(* Logix 5000 project; controller DUNEW2PLC1 vendor 1 type 14 code 221 rev 33.11; software revision 33.00; part 2 of 4 *)
(* tags used below, declared in another part *)
   LatchingTimeoutCounter : COUNTER;   // When you enter state 6 or 7, start counting seconds
   TimeoutTimer1 : TIMER;
   TimeoutTimer2 : TIMER;
   accel_xy : REAL;   // Tangential acceleration of the winding head in xy-plane
   ACTUATOR_POS : DINT;
   ALL_EOT_GOOD : BOOL;
   APA_IS_VERTICAL : BOOL;
   blink_off : TIMER;
   blink_on : TIMER;
   check_tension_stable : BOOL;   // Check if the tension is stable at the setpoint before moving the winding head
   ERROR_CODE : DINT;
   FRAME_LOC_FT_BTM : BOOL;
   FRAME_LOC_FT_MID : BOOL;
   FRAME_LOC_FT_TOP : BOOL;
   FRAME_LOC_HD_BTM : BOOL;
   FRAME_LOC_HD_MID : BOOL;
   FRAME_LOC_HD_TOP : BOOL;
   gamma : REAL;
   HEAD_POS : DINT;
   INIT_DONE : BOOL;
   J : REAL;
   MACHINE_SW_STAT : BOOL[32];
   MAS : BOOL;   // Motion Axis Stop
   MASTER_Z_GO : BOOL;
   MAX_TOLERABLE_Z : REAL;
   MCCD_X_Y_Axis1 : MOTION_INSTRUCTION;
   MINUS_X_EOT : BOOL;
   MINUS_Y_EOT : BOOL;
   MOVE_TYPE : INT;   // 0 = No Move 1 = XY JOG 2 = XY Plane Move 3 = Z JOG 4 = Z Axis Move 5 = Toggle Latch Actuator 6 = Home the Latch Actuator
   NEXTSTATE : DINT;
   PLUS_X_EOT : BOOL;
   PLUS_Y_EOT : BOOL;
   ResetPB : BOOL;
   Safety_Tripped_S : BOOL;
   speed_regulator_switch : BOOL;   // This is our "enable safe speed" switch, repurposed to switch the speed regulator
   STATE : DINT;   // CURRENT State Machine State
   T01 : TIMER;
   tension : ALIAS FOR Local:4:I.Ch01.Data;   // wire tension (N)
   TENSION_CONTROL_OK : BOOL;
   TENSION_ON_SWITCH : BOOL;
   tension_stable_timer : TIMER;
   v_0 : REAL;
   v_xy : REAL;   // velocity of winding head in xy plane
   v_xyz : REAL;   // Velocity of winding head in xyz space
   wire_break_proxy : BOOL;
   wire_break_tension : REAL;
   X_axis : AXIS_CIP_DRIVE;
   X_PARKED : BOOL;
   X_POSITION : ALIAS FOR POSITION[0,0];
   X_XFER_OK : BOOL;   // If at the head, check head support arms. Same for foot
   X_Y : COORDINATE_SYSTEM;
   XY_ACCELERATION : REAL;   // Maximum positive acceleration for position move.
   XY_DECELERATION : REAL;   // Maximum negative acceleration for position move.
   XY_SPEED : REAL;   // Maximum velocity for position move.
   XY_SPEED_REQ : REAL;   // XY Requested speed copy of XY_Speed to be used for MCLM and MCCD in MoveXY
   Y_axis : AXIS_CIP_DRIVE;
   Y_MOUNT_XFER_OK : BOOL;
   Y_POSITION : ALIAS FOR POSITION[0,1];
   Y_XFER_OK : BOOL;
   Y_Xfer_Window_Btm : BOOL;
   Y_Xfer_Window_Mid : BOOL;
   Y_Xfer_Window_Top : BOOL;
   Z_axis : AXIS_CIP_DRIVE;
   Z_EOT : BOOL;
   Z_EXTENDED : BOOL;
   Z_FIXED_LATCHED : BOOL;
   Z_FIXED_PRESENT : BOOL;
   Z_RETRACTED : BOOL;
   Z_STAGE_LATCHED : BOOL;
   Z_STAGE_PRESENT : BOOL;   // Winding head is on the Z-arm
(* Latch_UnLatch_State_6_7_8, continued *)

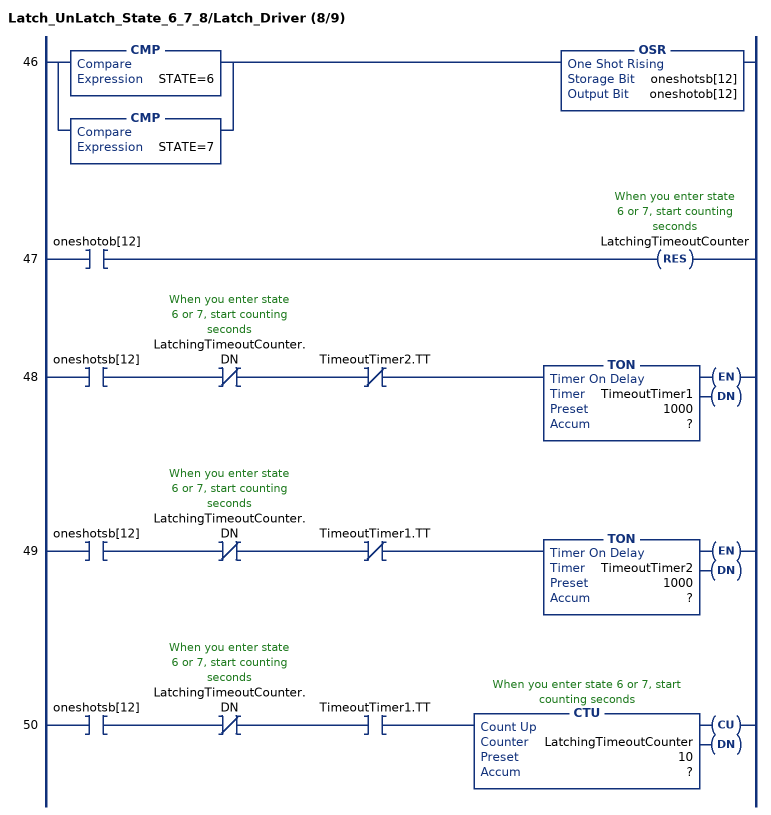
   [picture p24: Latch_UnLatch_State_6_7_8/Latch_Driver rungs 46-50]
   46: [CMP(STATE=6) ,CMP(STATE=7) ]OSR(oneshotsb[12],oneshotob[12]);
   47: XIC(oneshotob[12])RES(LatchingTimeoutCounter);
   48: XIC(oneshotsb[12])XIO(LatchingTimeoutCounter.DN)XIO(TimeoutTimer2.TT)TON(TimeoutTimer1,?,?);
   49: XIC(oneshotsb[12])XIO(LatchingTimeoutCounter.DN)XIO(TimeoutTimer1.TT)TON(TimeoutTimer2,?,?);
   50: XIC(oneshotsb[12])XIO(LatchingTimeoutCounter.DN)XIC(TimeoutTimer1.TT)CTU(LatchingTimeoutCounter,?,?);
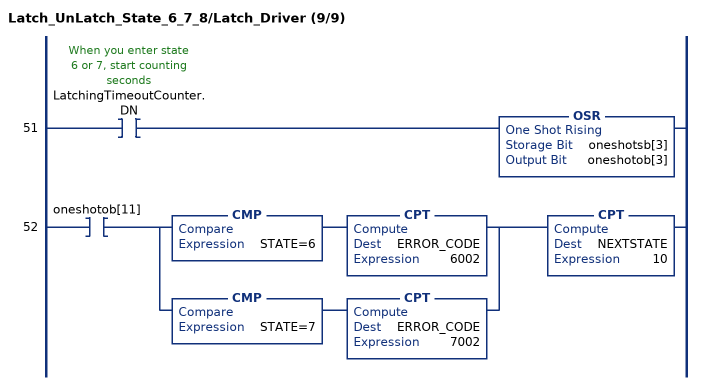
   51: XIC(LatchingTimeoutCounter.DN)OSR(oneshotsb[3],oneshotob[3]);
   52: XIC(oneshotob[11])[CMP(STATE=6) CPT(ERROR_CODE,6002) ,CMP(STATE=7) CPT(ERROR_CODE,7002) ]CPT(NEXTSTATE,10);
END_ROUTINE
END_PROGRAM

PROGRAM MainProgram   (* main routine MainRoutine *)
VAR
   Z_RETRACTED_1A : BOOL := 1; {access Read Only}
   Z_RETRACTED_1B : BOOL := 1; {access Read Only}
   Z_RETRACTED_2A : BOOL := 1; {access Read Only}
   Z_RETRACTED_2B : BOOL := 1; {access Read Only}
END_VAR

ROUTINE MainRoutine   (* ladder *)
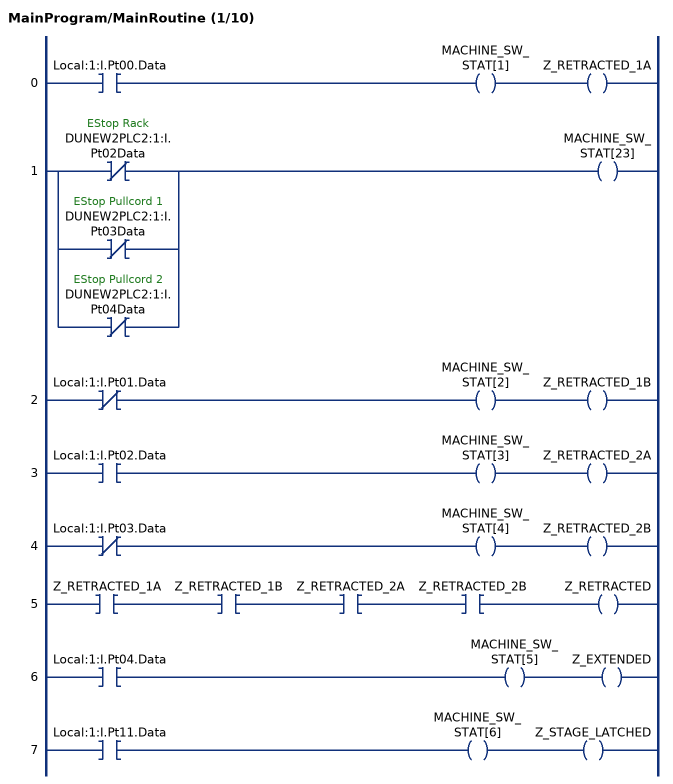
   0: XIC(Local:1:I.Pt00.Data)OTE(MACHINE_SW_STAT[1])OTE(Z_RETRACTED_1A);
   1: [XIO(DUNEW2PLC2:1:I.Pt02Data) ,[XIO(DUNEW2PLC2:1:I.Pt03Data) ,XIO(DUNEW2PLC2:1:I.Pt04Data) ] ]OTE(MACHINE_SW_STAT[23]);
   2: XIO(Local:1:I.Pt01.Data)OTE(MACHINE_SW_STAT[2])OTE(Z_RETRACTED_1B);
   3: XIC(Local:1:I.Pt02.Data)OTE(MACHINE_SW_STAT[3])OTE(Z_RETRACTED_2A);
   4: XIO(Local:1:I.Pt03.Data)OTE(MACHINE_SW_STAT[4])OTE(Z_RETRACTED_2B);
   5: XIC(Z_RETRACTED_1A)XIC(Z_RETRACTED_1B)XIC(Z_RETRACTED_2A)XIC(Z_RETRACTED_2B)OTE(Z_RETRACTED);
   6: XIC(Local:1:I.Pt04.Data)OTE(MACHINE_SW_STAT[5])OTE(Z_EXTENDED);
   7: XIC(Local:1:I.Pt11.Data)OTE(MACHINE_SW_STAT[6])OTE(Z_STAGE_LATCHED);
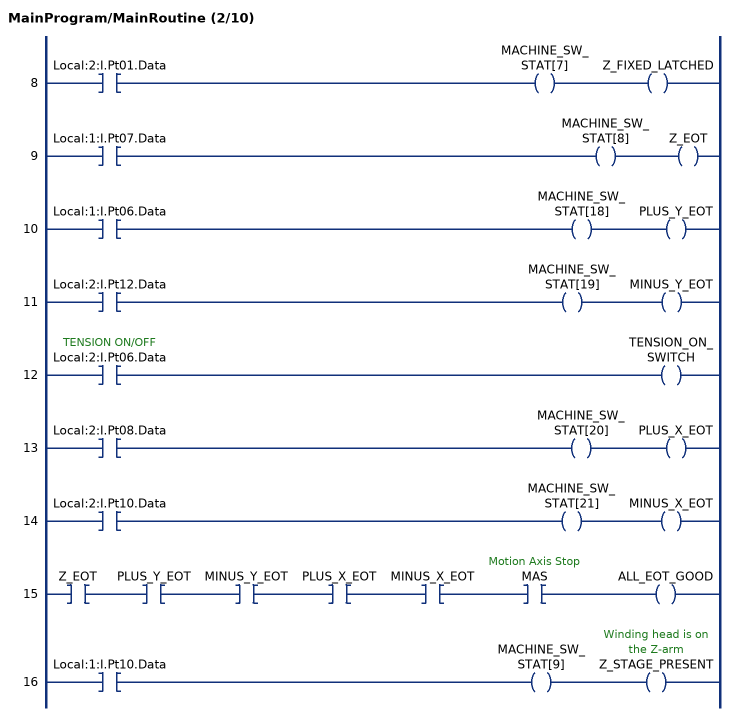
   8: XIC(Local:2:I.Pt01.Data)OTE(MACHINE_SW_STAT[7])OTE(Z_FIXED_LATCHED);
   9: XIC(Local:1:I.Pt07.Data)OTE(MACHINE_SW_STAT[8])OTE(Z_EOT);
   10: XIC(Local:1:I.Pt06.Data)OTE(MACHINE_SW_STAT[18])OTE(PLUS_Y_EOT);
   11: XIC(Local:2:I.Pt12.Data)OTE(MACHINE_SW_STAT[19])OTE(MINUS_Y_EOT);
   12: XIC(Local:2:I.Pt06.Data)OTE(TENSION_ON_SWITCH);
   13: XIC(Local:2:I.Pt08.Data)OTE(MACHINE_SW_STAT[20])OTE(PLUS_X_EOT);
   14: XIC(Local:2:I.Pt10.Data)OTE(MACHINE_SW_STAT[21])OTE(MINUS_X_EOT);
   15: XIC(Z_EOT)XIC(PLUS_Y_EOT)XIC(MINUS_Y_EOT)XIC(PLUS_X_EOT)XIC(MINUS_X_EOT)XIC(MAS)OTE(ALL_EOT_GOOD);
   16: XIC(Local:1:I.Pt10.Data)OTE(MACHINE_SW_STAT[9])OTE(Z_STAGE_PRESENT);
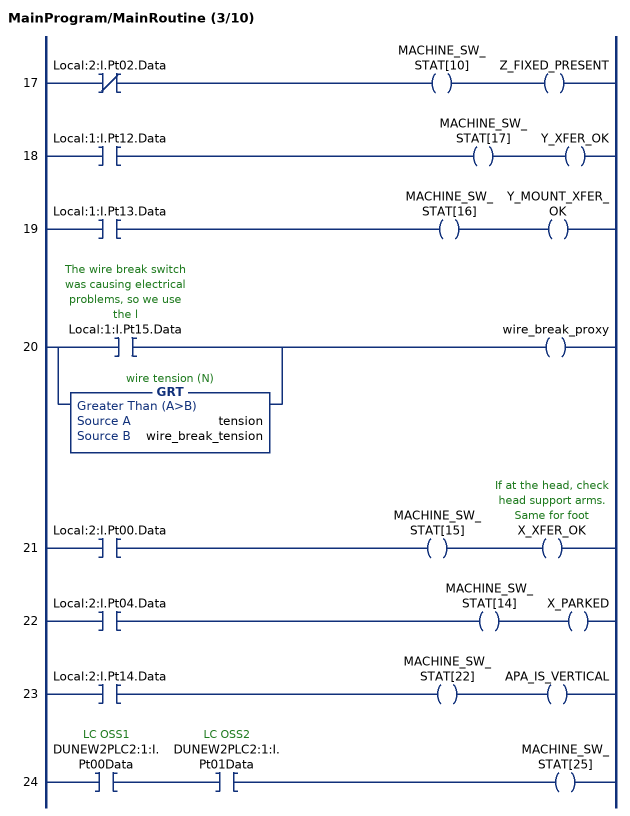
   17: XIO(Local:2:I.Pt02.Data)OTE(MACHINE_SW_STAT[10])OTE(Z_FIXED_PRESENT);
   18: XIC(Local:1:I.Pt12.Data)OTE(MACHINE_SW_STAT[17])OTE(Y_XFER_OK);
   19: XIC(Local:1:I.Pt13.Data)OTE(MACHINE_SW_STAT[16])OTE(Y_MOUNT_XFER_OK);
   20: [XIC(Local:1:I.Pt15.Data) ,GRT(tension,wire_break_tension) ]OTE(wire_break_proxy);
   21: XIC(Local:2:I.Pt00.Data)OTE(MACHINE_SW_STAT[15])OTE(X_XFER_OK);
   22: XIC(Local:2:I.Pt04.Data)OTE(MACHINE_SW_STAT[14])OTE(X_PARKED);
   23: XIC(Local:2:I.Pt14.Data)OTE(MACHINE_SW_STAT[22])OTE(APA_IS_VERTICAL);
   24: XIC(DUNEW2PLC2:1:I.Pt00Data)XIC(DUNEW2PLC2:1:I.Pt01Data)OTE(MACHINE_SW_STAT[25]);
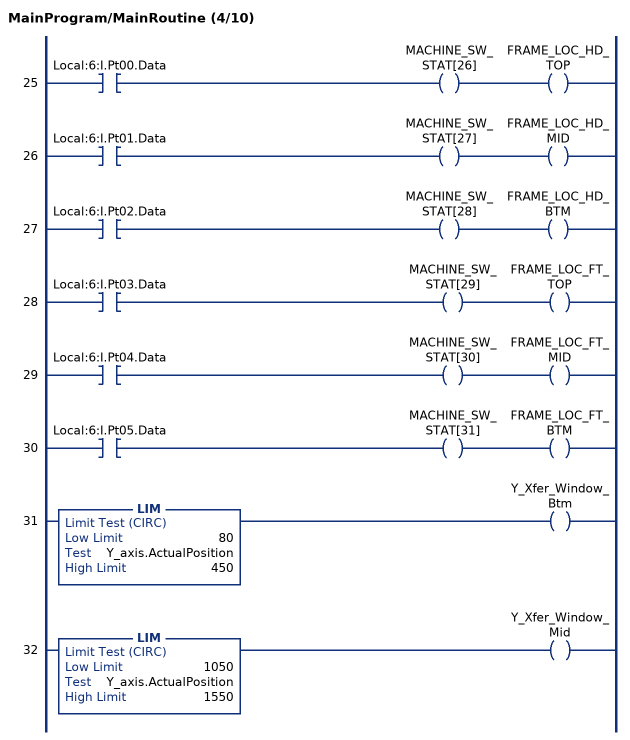
   25: XIC(Local:6:I.Pt00.Data)OTE(MACHINE_SW_STAT[26])OTE(FRAME_LOC_HD_TOP);
   26: XIC(Local:6:I.Pt01.Data)OTE(MACHINE_SW_STAT[27])OTE(FRAME_LOC_HD_MID);
   27: XIC(Local:6:I.Pt02.Data)OTE(MACHINE_SW_STAT[28])OTE(FRAME_LOC_HD_BTM);
   28: XIC(Local:6:I.Pt03.Data)OTE(MACHINE_SW_STAT[29])OTE(FRAME_LOC_FT_TOP);
   29: XIC(Local:6:I.Pt04.Data)OTE(MACHINE_SW_STAT[30])OTE(FRAME_LOC_FT_MID);
   30: XIC(Local:6:I.Pt05.Data)OTE(MACHINE_SW_STAT[31])OTE(FRAME_LOC_FT_BTM);
   31: LIM(80,Y_axis.ActualPosition,450)OTE(Y_Xfer_Window_Btm);
   32: LIM(1050,Y_axis.ActualPosition,1550)OTE(Y_Xfer_Window_Mid);
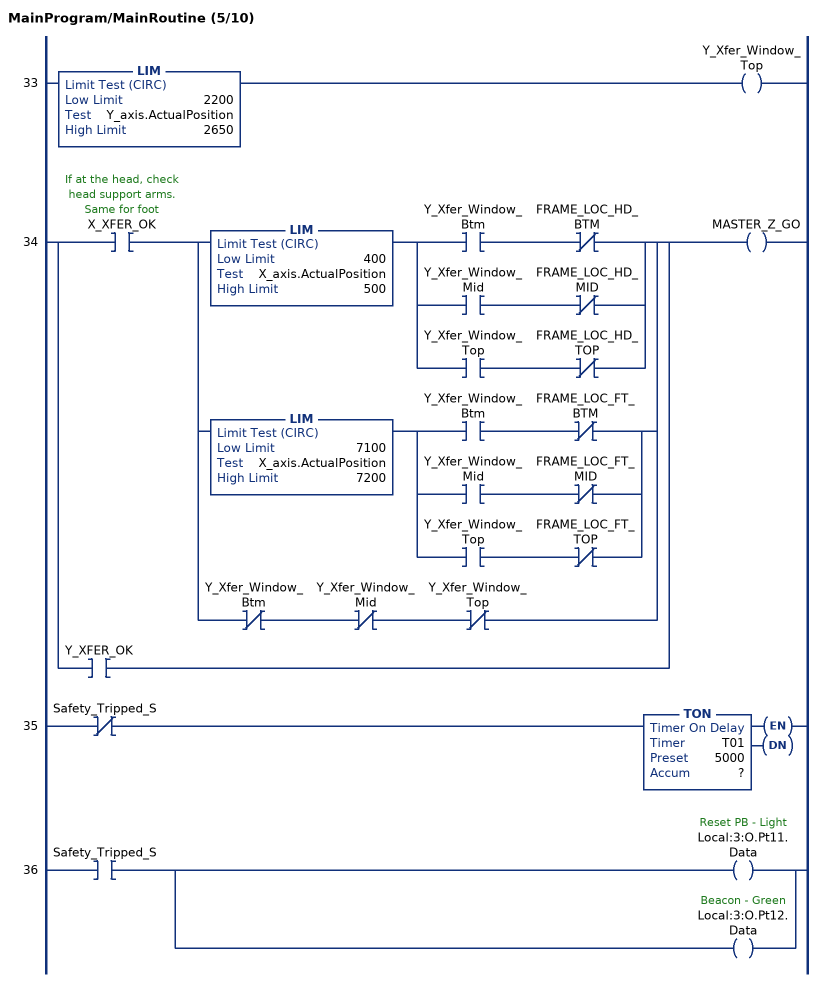
   33: LIM(2200,Y_axis.ActualPosition,2650)OTE(Y_Xfer_Window_Top);
   34: [XIC(X_XFER_OK) [LIM(400,X_axis.ActualPosition,500) [XIC(Y_Xfer_Window_Btm) XIO(FRAME_LOC_HD_BTM) ,XIC(Y_Xfer_Window_Mid) XIO(FRAME_LOC_HD_MID) ,XIC(Y_Xfer_Window_Top) XIO(FRAME_LOC_HD_TOP) ] ,LIM(7100,X_axis.ActualPosition,7200) [XIC(Y_Xfer_Window_Btm) XIO(FRAME_LOC_FT_BTM) ,XIC(Y_Xfer_Window_Mid) XIO(FRAME_LOC_FT_MID) ,XIC(Y_Xfer_Window_Top) XIO(FRAME_LOC_FT_TOP) ] ,XIO(Y_Xfer_Window_Btm) XIO(Y_Xfer_Window_Mid) XIO(Y_Xfer_Window_Top) ] ,XIC(Y_XFER_OK) ]OTE(MASTER_Z_GO);
   35: XIO(Safety_Tripped_S)TON(T01,?,?);
   36: XIC(Safety_Tripped_S)[OTE(Local:3:O.Pt11.Data) ,OTE(Local:3:O.Pt12.Data) ];
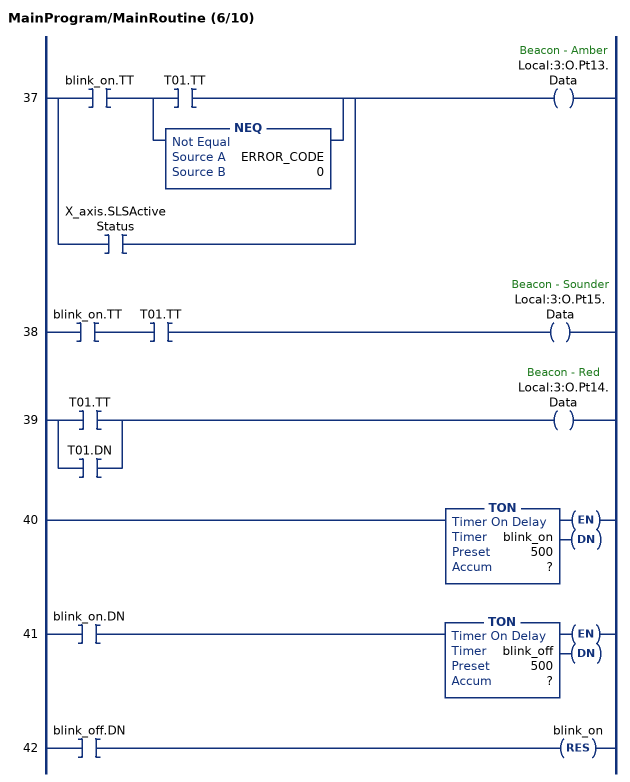
   37: [XIC(blink_on.TT) [XIC(T01.TT) ,NEQ(ERROR_CODE,0) ] ,XIC(X_axis.SLSActiveStatus) ]OTE(Local:3:O.Pt13.Data);
   38: XIC(blink_on.TT)XIC(T01.TT)OTE(Local:3:O.Pt15.Data);
   39: [XIC(T01.TT) ,XIC(T01.DN) ]OTE(Local:3:O.Pt14.Data);
   40: TON(blink_on,?,?);
   41: XIC(blink_on.DN)TON(blink_off,?,?);
   42: XIC(blink_off.DN)RES(blink_on);
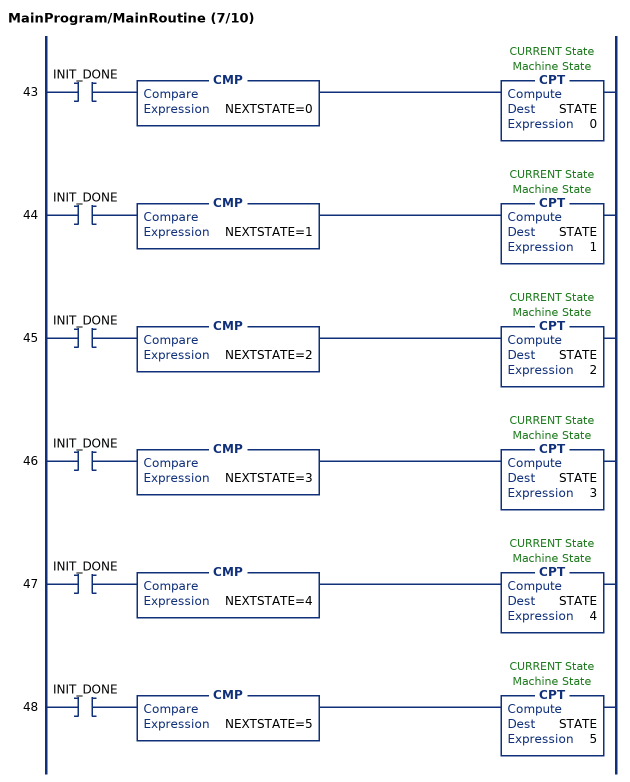
   43: XIC(INIT_DONE)CMP(NEXTSTATE=0)CPT(STATE,0);
   44: XIC(INIT_DONE)CMP(NEXTSTATE=1)CPT(STATE,1);
   45: XIC(INIT_DONE)CMP(NEXTSTATE=2)CPT(STATE,2);
   46: XIC(INIT_DONE)CMP(NEXTSTATE=3)CPT(STATE,3);
   47: XIC(INIT_DONE)CMP(NEXTSTATE=4)CPT(STATE,4);
   48: XIC(INIT_DONE)CMP(NEXTSTATE=5)CPT(STATE,5);
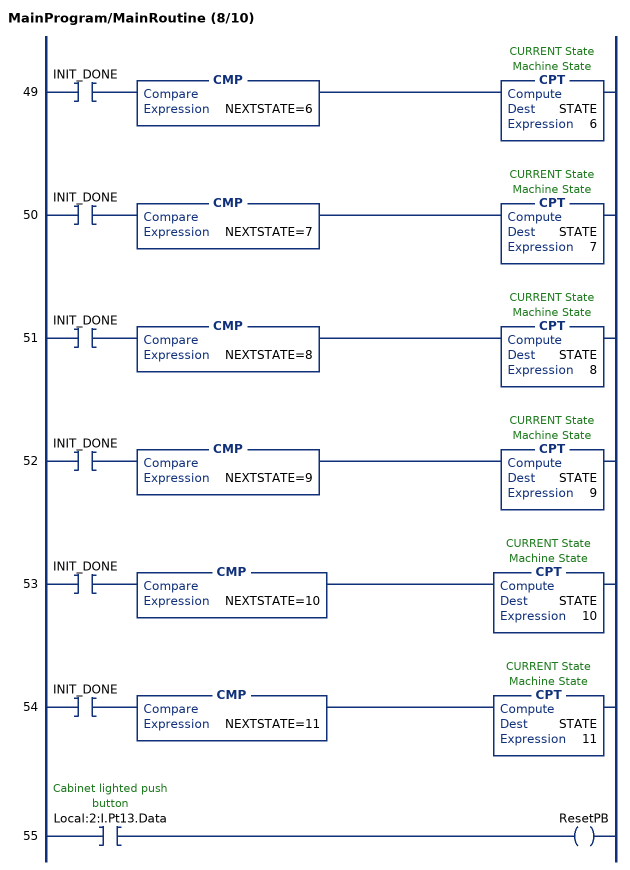
   49: XIC(INIT_DONE)CMP(NEXTSTATE=6)CPT(STATE,6);
   50: XIC(INIT_DONE)CMP(NEXTSTATE=7)CPT(STATE,7);
   51: XIC(INIT_DONE)CMP(NEXTSTATE=8)CPT(STATE,8);
   52: XIC(INIT_DONE)CMP(NEXTSTATE=9)CPT(STATE,9);
   53: XIC(INIT_DONE)CMP(NEXTSTATE=10)CPT(STATE,10);
   54: XIC(INIT_DONE)CMP(NEXTSTATE=11)CPT(STATE,11);
   55: XIC(Local:2:I.Pt13.Data)OTE(ResetPB);
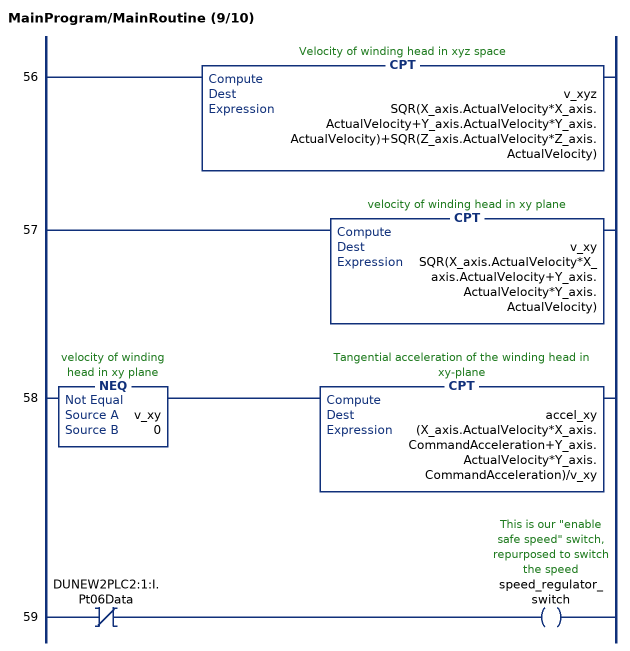
   56: CPT(v_xyz,SQR(X_axis.ActualVelocity*X_axis.ActualVelocity+Y_axis.ActualVelocity*Y_axis.ActualVelocity)+SQR(Z_axis.ActualVelocity*Z_axis.ActualVelocity));
   57: CPT(v_xy,SQR(X_axis.ActualVelocity*X_axis.ActualVelocity+Y_axis.ActualVelocity*Y_axis.ActualVelocity));
   58: NEQ(v_xy,0)CPT(accel_xy,(X_axis.ActualVelocity*X_axis.CommandAcceleration+Y_axis.ActualVelocity*Y_axis.CommandAcceleration)/v_xy);
   59: XIO(DUNEW2PLC2:1:I.Pt06Data)OTE(speed_regulator_switch);
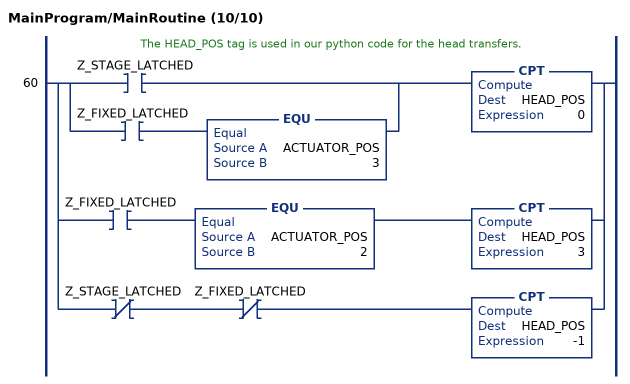
   // The HEAD_POS tag is used in our python code for the head transfers.
   60: [[XIC(Z_STAGE_LATCHED) ,XIC(Z_FIXED_LATCHED) EQU(ACTUATOR_POS,3) ] CPT(HEAD_POS,0) ,XIC(Z_FIXED_LATCHED) EQU(ACTUATOR_POS,2) CPT(HEAD_POS,3) ,XIO(Z_STAGE_LATCHED) XIO(Z_FIXED_LATCHED) CPT(HEAD_POS,-1) ];
END_ROUTINE
END_PROGRAM

PROGRAM MoveXY_State_2_3   (* main routine MoveXY *)
VAR
   d_raw : REAL;
   dx : REAL := 0.0039;
   dy : REAL := 0.0017;
   eot_triggered : BOOL;
   k : REAL := 211538.47;
   max_integral : DINT := 1000;
   min_integral : DINT := -1000;
   min_regulated_speed : DINT := 100;
   near_ending : BOOL;   // True if distance to xy-move target is less than the required stopping distance
   near_ending_trigger : BOOL;
   oneshotob : BOOL[32];
   oneshotsb : BOOL[32] := ([2] := 1, [4] := 1, [11] := 1, [12] := 1, [13] := 1, [14] := 1, [15] := 1, [16] := 1, [17] := 1);
   regulated_speed : REAL := 899.9713;
   regulator_loop_timer : TIMER := (PRE := 1);
   speed_set_to_zero : BOOL;
   speed_tension_setpoint : REAL := 8.5;
   starting_x : REAL := -0.0039;
   starting_y : REAL := -0.0017;
   STATE3_IND : BOOL; {access Read Only}
   stopping_distance : REAL;   // Calculate the distance required to perform a jerk-limited stop at the gurrent jerk, acceleration, and speed
   stopping_ratio : REAL := 0.2532453;
   trigger_xy_move : BOOL;
   v_max : REAL := 899.9713;
   x_dist_to_target : REAL := 0.6653;
   X_max_speed : REAL := 825.0; {constant}
   x_time : REAL := 211538.47;
   xy_accel_jerk : DINT := 1500;
   XY_AXIS_STAT : MOTION_INSTRUCTION[32] := ([2].FLAGS := 536870912, [2].DN := 1, [3].FLAGS := 536870912, [3].DN := 1, [4].FLAGS := 33554432, [5].FLAGS := 33554432, [6].FLAGS := 704643072, [6].DN := 1, [6].PC := 1);
   xy_d_alpha : REAL := 1.0;
   xy_d_dt : DINT := 50;
   xy_d_term : REAL;
   xy_d_term_prev : REAL;
   xy_d_timer : TIMER := (PRE := 50);
   xy_decel_jerk : DINT := 2000;
   xy_default_speed : DINT;
   xy_dist_to_target : REAL := 0.66530246;
   xy_dt : DINT := 1;
   xy_error : REAL := 6.0954127;
   xy_error_prev : REAL := 6.0985594;
   xy_i_term : REAL := 900.0352;
   xy_kd : REAL;
   xy_ki : REAL := 300.0;
   xy_kp : REAL;
   xy_p_term : REAL;
   XY_POS_LOCK_STAT : BOOL; {access Read Only}
   y_dist_to_target : REAL := -0.0018;
   Y_max_speed : REAL := 600.0; {constant}
   y_time : REAL := 352941.16;
END_VAR

ROUTINE MoveXY   (* ladder *)
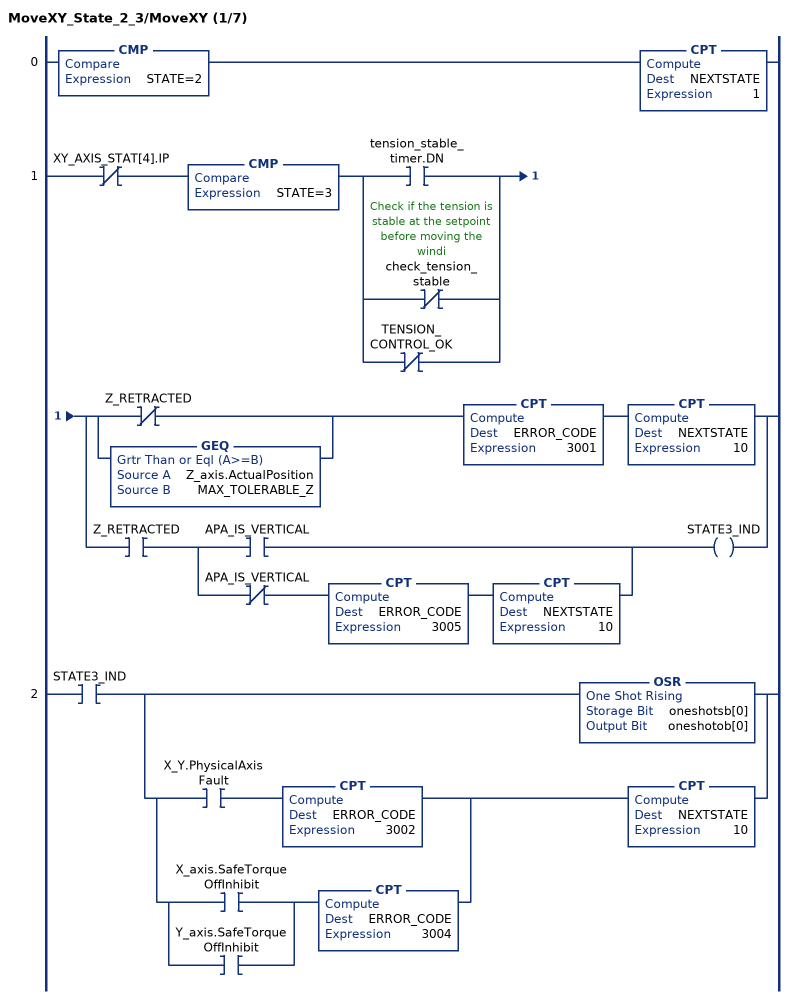
   0: CMP(STATE=2)CPT(NEXTSTATE,1);
   1: XIO(XY_AXIS_STAT[4].IP)CMP(STATE=3)[XIC(tension_stable_timer.DN) ,XIO(check_tension_stable) ,XIO(TENSION_CONTROL_OK) ][[XIO(Z_RETRACTED) ,GEQ(Z_axis.ActualPosition,MAX_TOLERABLE_Z) ] CPT(ERROR_CODE,3001) CPT(NEXTSTATE,10) ,XIC(Z_RETRACTED) [XIC(APA_IS_VERTICAL) ,XIO(APA_IS_VERTICAL) CPT(ERROR_CODE,3005) CPT(NEXTSTATE,10) ] OTE(STATE3_IND) ];
   2: XIC(STATE3_IND)[OSR(oneshotsb[0],oneshotob[0]) ,[XIC(X_Y.PhysicalAxisFault) CPT(ERROR_CODE,3002) ,[XIC(X_axis.SafeTorqueOffInhibit) ,XIC(Y_axis.SafeTorqueOffInhibit) ] CPT(ERROR_CODE,3004) ] CPT(NEXTSTATE,10) ];
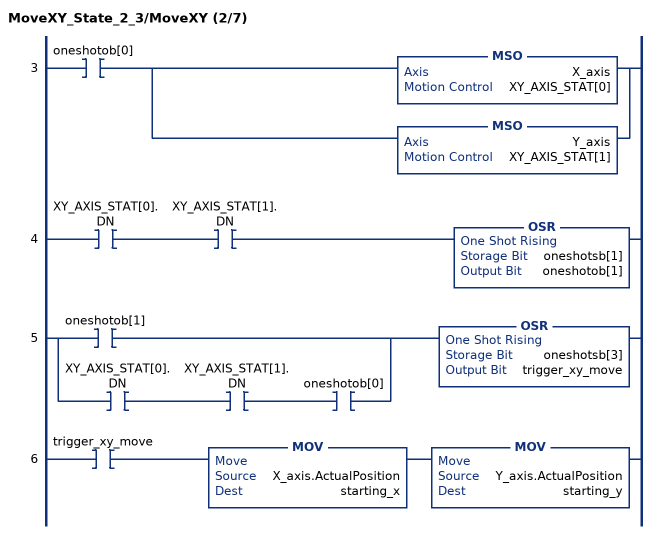
   3: XIC(oneshotob[0])[MSO(X_axis,XY_AXIS_STAT[0]) ,MSO(Y_axis,XY_AXIS_STAT[1]) ];
   4: XIC(XY_AXIS_STAT[0].DN)XIC(XY_AXIS_STAT[1].DN)OSR(oneshotsb[1],oneshotob[1]);
   5: [XIC(oneshotob[1]) ,XIC(XY_AXIS_STAT[0].DN) XIC(XY_AXIS_STAT[1].DN) XIC(oneshotob[0]) ]OSR(oneshotsb[3],trigger_xy_move);
   6: XIC(trigger_xy_move)MOV(X_axis.ActualPosition,starting_x)MOV(Y_axis.ActualPosition,starting_y);
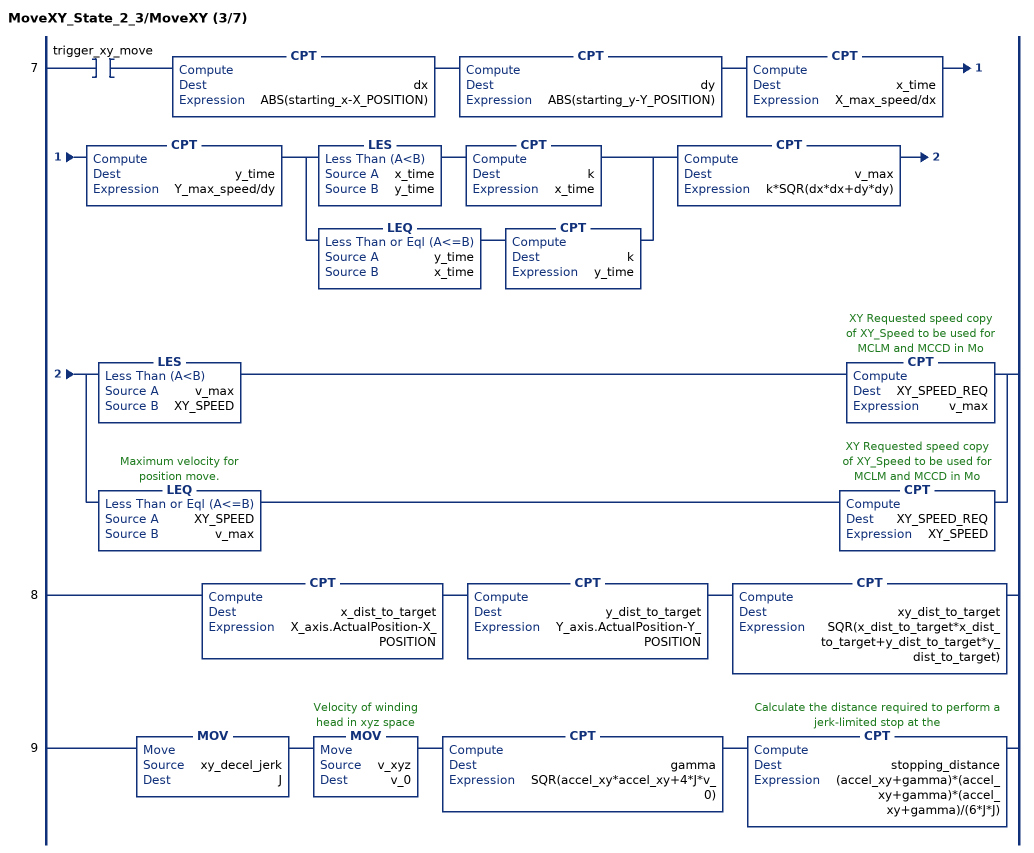
   7: XIC(trigger_xy_move)CPT(dx,ABS(starting_x-X_POSITION))CPT(dy,ABS(starting_y-Y_POSITION))CPT(x_time,X_max_speed/dx)CPT(y_time,Y_max_speed/dy)[LES(x_time,y_time) CPT(k,x_time) ,LEQ(y_time,x_time) CPT(k,y_time) ]CPT(v_max,k*SQR(dx*dx+dy*dy))[LES(v_max,XY_SPEED) CPT(XY_SPEED_REQ,v_max) ,LEQ(XY_SPEED,v_max) CPT(XY_SPEED_REQ,XY_SPEED) ];
   8: CPT(x_dist_to_target,X_axis.ActualPosition-X_POSITION)CPT(y_dist_to_target,Y_axis.ActualPosition-Y_POSITION)CPT(xy_dist_to_target,SQR(x_dist_to_target*x_dist_to_target+y_dist_to_target*y_dist_to_target));
   9: MOV(xy_decel_jerk,J)MOV(v_xyz,v_0)CPT(gamma,SQR(accel_xy*accel_xy+4*J*v_0))CPT(stopping_distance,(accel_xy+gamma)*(accel_xy+gamma)*(accel_xy+gamma)/(6*J*J));
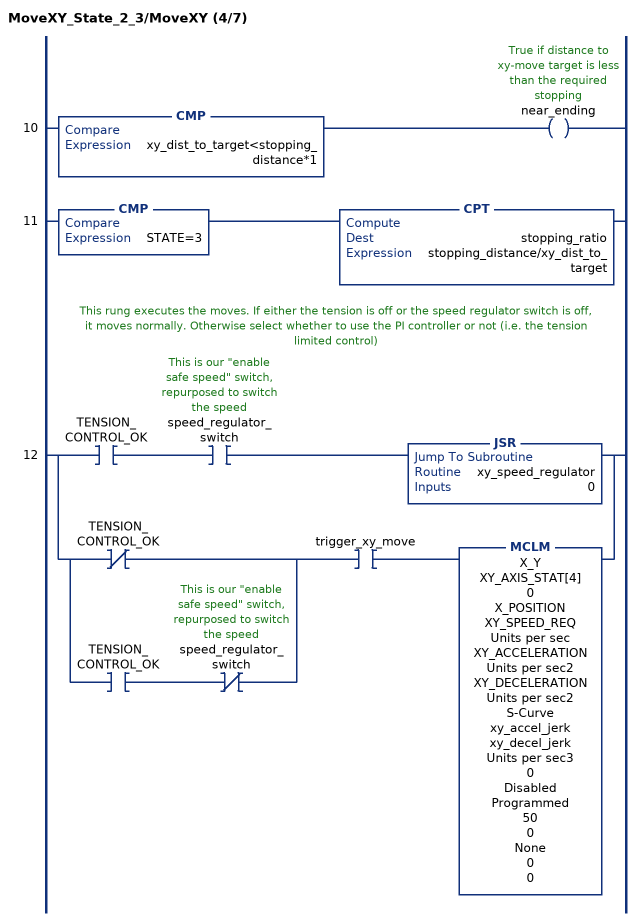
   10: CMP(xy_dist_to_target<stopping_distance*1)OTE(near_ending);
   11: CMP(STATE=3)CPT(stopping_ratio,stopping_distance/xy_dist_to_target);
   // This rung executes the moves. If either the tension is off or the speed regulator switch is off, it moves normally. Otherwise select whether to use the PI controller or not (i.e. the tension limited control)
   12: [XIC(TENSION_CONTROL_OK) XIC(speed_regulator_switch) JSR(xy_speed_regulator,0) ,[XIO(TENSION_CONTROL_OK) ,XIC(TENSION_CONTROL_OK) XIO(speed_regulator_switch) ] XIC(trigger_xy_move) MCLM(X_Y,XY_AXIS_STAT[4],0,X_POSITION,XY_SPEED_REQ,Units per sec,XY_ACCELERATION,Units per sec2,XY_DECELERATION,Units per sec2,S-Curve,xy_accel_jerk,xy_decel_jerk,Units per sec3,0,Disabled,Programmed,50,0,None,0,0) ];
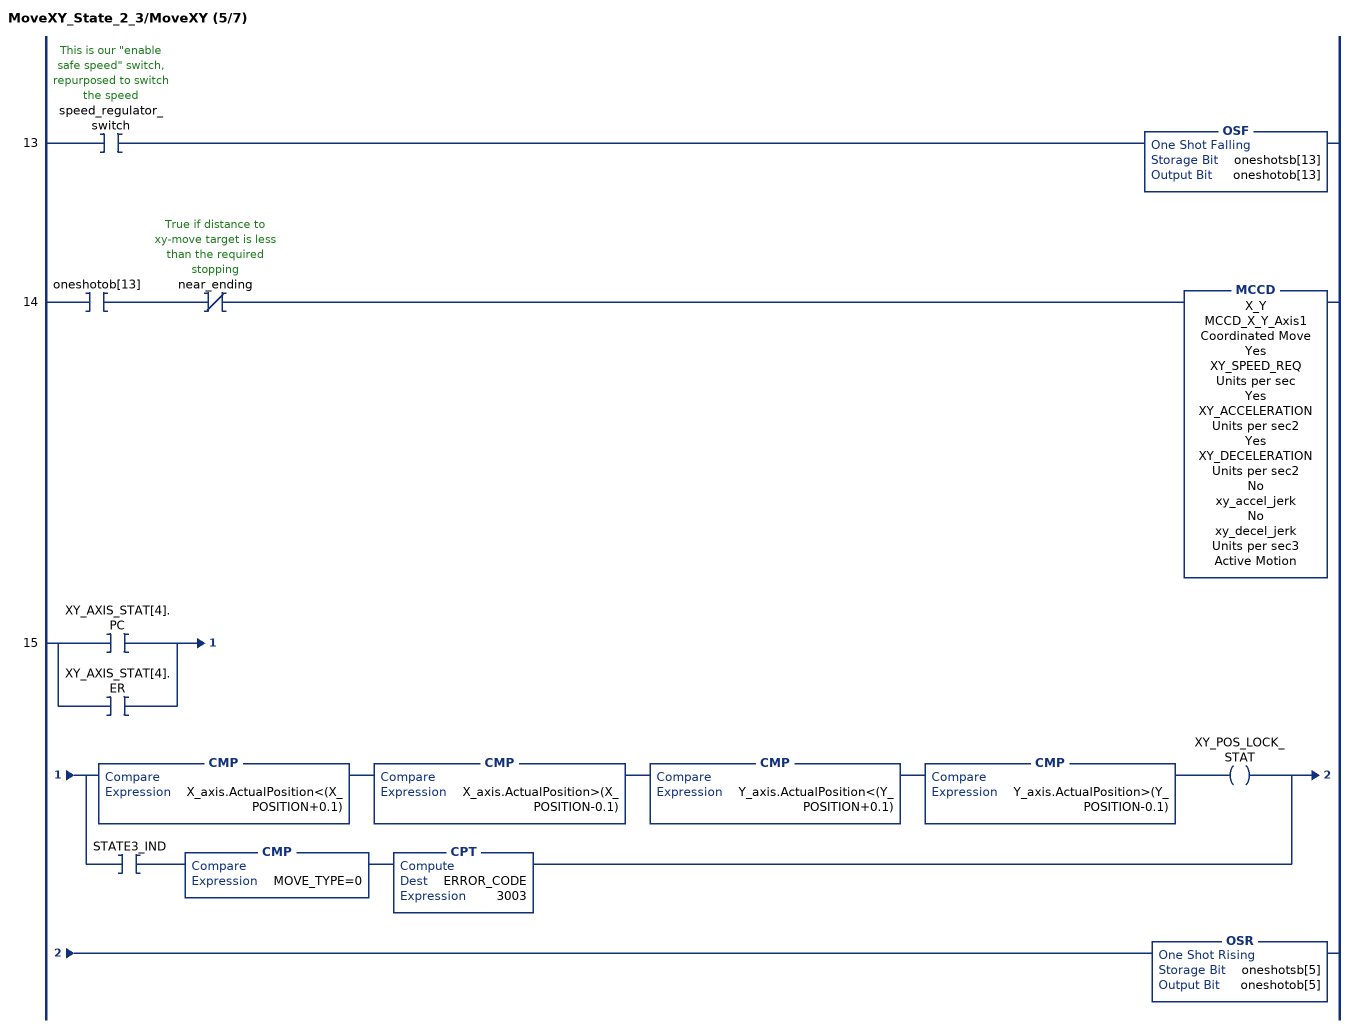
   13: XIC(speed_regulator_switch)OSF(oneshotsb[13],oneshotob[13]);
   14: XIC(oneshotob[13])XIO(near_ending)MCCD(X_Y,MCCD_X_Y_Axis1,Coordinated Move,Yes,XY_SPEED_REQ,Units per sec,Yes,XY_ACCELERATION,Units per sec2,Yes,XY_DECELERATION,Units per sec2,No,xy_accel_jerk,No,xy_decel_jerk,Units per sec3,Active Motion);
   15: [XIC(XY_AXIS_STAT[4].PC) ,XIC(XY_AXIS_STAT[4].ER) ][CMP(X_axis.ActualPosition<(X_POSITION+0.1)) CMP(X_axis.ActualPosition>(X_POSITION-0.1)) CMP(Y_axis.ActualPosition<(Y_POSITION+0.1)) CMP(Y_axis.ActualPosition>(Y_POSITION-0.1)) OTE(XY_POS_LOCK_STAT) ,XIC(STATE3_IND) CMP(MOVE_TYPE=0) CPT(ERROR_CODE,3003) ]OSR(oneshotsb[5],oneshotob[5]);
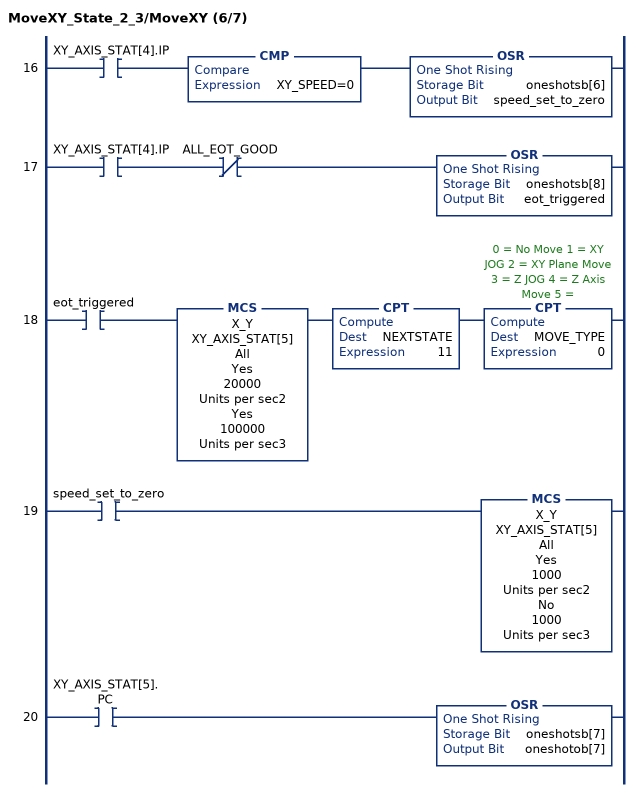
   16: XIC(XY_AXIS_STAT[4].IP)CMP(XY_SPEED=0)OSR(oneshotsb[6],speed_set_to_zero);
   17: XIC(XY_AXIS_STAT[4].IP)XIO(ALL_EOT_GOOD)OSR(oneshotsb[8],eot_triggered);
   18: XIC(eot_triggered)MCS(X_Y,XY_AXIS_STAT[5],All,Yes,20000,Units per sec2,Yes,100000,Units per sec3)CPT(NEXTSTATE,11)CPT(MOVE_TYPE,0);
   19: XIC(speed_set_to_zero)MCS(X_Y,XY_AXIS_STAT[5],All,Yes,1000,Units per sec2,No,1000,Units per sec3);
   20: XIC(XY_AXIS_STAT[5].PC)OSR(oneshotsb[7],oneshotob[7]);
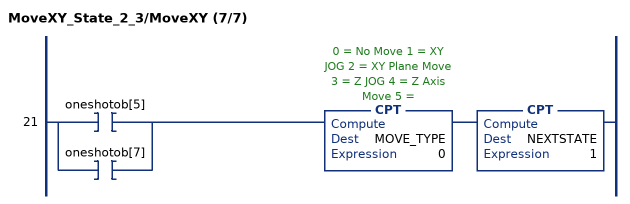
   21: [XIC(oneshotob[5]) ,XIC(oneshotob[7]) ]CPT(MOVE_TYPE,0)CPT(NEXTSTATE,1);
END_ROUTINE
